FUNCTION_BLOCK forgettingFactor
VAR_INPUT
	inputValue : REAL;
END_VAR
VAR_OUTPUT
	meanValue : REAL;
END_VAR
VAR
	A_Factor : REAL := 0.5;
	y_um :REAL;
	meanValue_um : REAL;
END_VAR

meanValue := A_Factor * meanValue_um + (1-A_Factor)*y_um;

y_um := inputValue;
meanValue_um := meanValue;

END_FUNCTION_BLOCK

(* stored: Version 1.1.0.1, ProductVersion 3.1.4024.13
   POU forgettingFactor: Id {850b9e85-df92-4a3b-94bb-e188e3082866}, SpecialFunc None *)
